// TIA Portal V19 export
VAR_GLOBAL   // PLC tag table "U3Em1"
END_VAR
VAR_GLOBAL CONSTANT   // user constants
   U3EM1_NO_OF_AXES : USInt := 1;   // Starts with 1. E.g., the value 4 means that 4 axes exist.
   NO_JOB : Int := 0;
   U3EM1_JOB_STARTING : Int := 100;
   U3EM1_JOB_POS_MOVING : Int := 200;
   U3EM1_JOB_HOLODING : Int := 300;
   MATERIAL_DETECTION_UPPER_OneUnit : DInt := 4;
   U3EM1_JOB_RESETING : Int := 400;
   U3EM1_JOB_HOMING : Int := 500;
   U3EM1_JOB_STOPPING : Int := 600;
   U3EM1_JOB_UNHLODING : Int := 700;
   U3EM1_JOB_SPECIALFUNC_ABSPOS : Int := 800;
END_VAR
